(*
  Base camera system
  Implements I_Camera: set I_CameraSink.   
*)
FUNCTION_BLOCK ABSTRACT FB_CameraBase EXTENDS FB_Commons IMPLEMENTS I_Camera, I_CameraTriggerDevice

VAR
  _bInitialized             : BOOL;
  _iCameraSink              : I_CameraSink;
  _iCameraTrigger           : I_CameraTrigger;
  _bSimulate                : BOOL;
  _nPrintUnitResolution     : UDINT;           (*printhead pixel resolution [dpi]*)
  _nPrintUnitSubPx          : UDINT;           (*print unit SubPixel resolution [SubPx]*)
  _bUseCameraTrigger        : BOOL;            (*use a trigger output timestamp I/O*)
  _bUseCameraTriggerFeedback : BOOL;           (*use a camera triggered feedback timestamp I/O*)
  _eCameraMode              : E_CameraMode;    (*desired camera mode*)
  _ePossibleMode            : E_CameraMode;    (*currently possible mode*)
  _fSubstrateLength         : LREAL := 1;      (*Substrate length [m]*)
  _fSubstrateWidth          : LREAL := 1;      (*Substrate width [m]*)
  _fImageLength             : LREAL := 1;      (*Image length [m]*)
  _fImageWidth              : LREAL := 1;      (*Image width [m]*)
  _fFrameLength             : LREAL := 1;      (*Camera Frame width in [px]*)
  _bActivated               : BOOL;            (*Camera is activated*)
  _sVisuName                : STRING := 'unvailable';     (*detail visualisation instance name*)
  
  // status
  _bCamTriggerOk            : BOOL;
  _bCamTriggerStarted       : BOOL;
  _bCamTriggerDone          : BOOL;   
  _nCamStartPos             : DINT;            (*Cam start position ideal [SubPx]*)
  _nCamStartPosDeviation    : DINT;            (*Cam stated position real [SubPx]*)
  _nRxCamPoints             : UDINT;           (*number of received cam points*)

  // helper
  stCamPoint                : ST_DeformationPointAccurate;(*actual camera point*)
    
  // messaging
  _pMsgConfig               : POINTER TO CalmarCommons.ST_MSG_CONFIG;
END_VAR

VAR PERSISTENT
  _fTriggerDistance         : LREAL;           (*[m] Distance between Sensor and Trigger*)
  _fTriggerPulseLength      : LREAL := 10;     (*[ms] Length of trigger signal in ms, min. 3 bus cycles*)
  _fDetectToCameraOffset    : LREAL := 0.1;    (*[m] Distance between input trigger and camera, mech.*)
  _fCameraToPrintOffset     : LREAL := 0.0;    (*[m] Distance between Camera and PU, mech, This offset can be used to shift the reference of a camera/sheet-detect, e.g. because this reference is different from to one where the alignment Camera/sheetdetect-PrintUnit has been made*)
END_VAR

METHOD ActivateCam : BOOL
VAR_INPUT
  iCameraSink : I_CameraSink;
END_VAR
IF iCameraSink = 0 THEN
  LogError('Invalid parameter (0 pointer)');
  ActivateCam := FALSE;
  RETURN; 
ELSIF _iCameraSink <> 0 AND iCameraSink <>_iCameraSink THEN
  LogError('SetSink failed: other sink already exists');
  ActivateCam := FALSE;
  RETURN; 
END_IF 

_iCameraSink := iCameraSink;
_iCameraTrigger.Enable(iCam:=THIS^, bUseCameraTrigger:=_bUseCameraTrigger, bUseCameraTriggerFeedback:=_bUseCameraTriggerFeedback);

_bActivated := TRUE;
ActivateCam:=TRUE;
END_METHOD

(*
  Activate/Deactivate camera trigger device
*)
PROPERTY bEnableTrigger : BOOL
SET
IF bEnableTrigger THEN
  _iCameraTrigger.Enable(iCam := THIS^, bUseCameraTrigger:= _bUseCameraTrigger, bUseCameraTriggerFeedback:=_bUseCameraTriggerFeedback);
ELSE
  _iCameraTrigger.Disable();
END_IF
END_SET
END_PROPERTY

(*
  Activate/Deactivate camera manual teach mode
*)
PROPERTY bManualTeach : BOOL
SET
_iCameraTrigger.bManualTeach := bManualTeach;
END_SET
END_PROPERTY

{attribute 'monitoring':='call'}
PROPERTY bSimulate : BOOL
GET
bSimulate := _bSimulate;
END_GET
SET
_bSimulate := bSimulate;
END_SET
END_PROPERTY

METHOD CamTrigger
VAR_INPUT
  bOk             : BOOL;     // trigger is ok
	nPos            : DINT;     // camera triggered position
  nPosDeviation   : DINT;     // camera started deviation
  nX0             : DINT;     // detected position sheet/repetition
END_VAR
_nRxCamPoints := 0;
_bCamTriggerStarted    := TRUE;
_bCamTriggerDone       := FALSE;
_bCamTriggerOk  := bOk;
_nCamStartPos   := nPos;
_nCamStartPosDeviation := nPosDeviation;

LogLvl(Lvl:=E_LogSeverity.Debug, Msg:=F_Concat2('CamTrigger at X0=', TO_STRING(nPos)));
IF _iCameraSink <> 0 THEN   // inform sink
  _iCameraSink.CamStarted(nX0:=nX0);
END_IF
END_METHOD

METHOD CamTriggerDone
_bCamTriggerStarted    := FALSE;  // this call marks the end of the camera trigger period
_bCamTriggerDone       := TRUE;

LogLvl(Lvl:=E_LogSeverity.Debug, Msg:='CamTriggerDone');
IF _iCameraSink <> 0 THEN   // inform sink
  _iCameraSink.CamDone();
END_IF
END_METHOD

METHOD DeactivateCam : BOOL
VAR_INPUT
  iSink : I_CameraSink;
END_VAR
IF _iCameraSink <> 0 AND iSink <> _iCameraSink THEN
  LogError('remove sink failed: inconsistent');
  DeactivateCam := FALSE;
  RETURN;  
END_IF

_iCameraSink := 0;
_iCameraTrigger.Disable();
_bActivated := FALSE;
DeactivateCam:=TRUE;
END_METHOD

{attribute 'monitoring':='call'}
PROPERTY ABSTRACT eCameraMode : E_CameraMode
GET
END_GET
END_PROPERTY

{attribute 'monitoring':='call'}
PROPERTY ABSTRACT eDeviceType : E_CameraDevice
GET
END_GET
END_PROPERTY

{attribute 'monitoring':='call'}
PROPERTY fCameraToPrintOffset : LREAL
GET
//This offset can be used to shift the reference of a camera, e.g. because this reference is different from to one where the alignment Camera-PrintUnit has been made
fCameraToPrintOffset := _fCameraToPrintOffset;
END_GET
SET
_fCameraToPrintOffset := fCameraToPrintOffset;
END_SET
END_PROPERTY

{attribute 'monitoring':='call'}
PROPERTY fDetectToCameraOffset : LREAL
GET
//This offset can be used to shift the reference of a camera, e.g. because this reference is different from to one where the alignment Camera-PrintUnit has been made
fDetectToCameraOffset := _fDetectToCameraOffset;
END_GET
SET
_fDetectToCameraOffset := fDetectToCameraOffset;
END_SET
END_PROPERTY

{attribute 'monitoring':='call'}
(* camera frame size in [px]*)
PROPERTY fFrameLength : LREAL
GET
fFrameLength := _fFrameLength;
END_GET
SET
_fFrameLength := fFrameLength;
END_SET
END_PROPERTY

{attribute 'monitoring':='call'}
(*Image Length/Depth in [m]*)
PROPERTY fImageLength : LREAL
GET
fImageLength := _fImageLength;
END_GET
SET
_fImageLength := fImageLength;
END_SET
END_PROPERTY

{attribute 'monitoring':='call'}
(*Image Width in [m]*)
PROPERTY fImageWidth : LREAL
GET
fImageWidth := _fImageWidth;
END_GET
SET
_fImageWidth := fImageWidth;
END_SET
END_PROPERTY

{attribute 'monitoring':='call'}
(*Substrate Length/Depth in [m]*)
PROPERTY fSubstrateLength : LREAL
GET
fSubstrateLength := _fSubstrateLength;
END_GET
SET
//ROI in Print direction
IF _iCameraTrigger <> 0 THEN
  _iCameraTrigger.SetSubstrateLength(fSubstrateLength := fSubstrateLength);   // save to camera trigger
  _fSubstrateLength := fSubstrateLength;                                      // save to camera
END_IF
END_SET
END_PROPERTY

{attribute 'monitoring':='call'}
(*Substrate Width in [m]*)
PROPERTY fSubstrateWidth : LREAL
GET
fSubstrateWidth := _fSubstrateWidth;
END_GET
SET
_fSubstrateWidth := fSubstrateWidth;
END_SET
END_PROPERTY

{attribute 'monitoring':='call'}
PROPERTY fTriggerDistance : LREAL
GET
fTriggerDistance := _fTriggerDistance;
END_GET
SET
_fTriggerDistance := fTriggerDistance;
END_SET
END_PROPERTY

PROPERTY fTriggerPulseLength : LREAL
GET
fTriggerPulseLength := _fTriggerPulseLength;
END_GET
END_PROPERTY

METHOD ABSTRACT GetCamStatus : BOOL
VAR_OUTPUT
  bConnectionOK  : BOOL;    // Camera connected
  bTeachOk       : BOOL;    // Teach successful
  nTeachedPoints : UDINT;   // Teached points for this job
  nScannedPoints : UDINT;   // Scanned points on current sheet  
  bCamStarted    : BOOL;    // Camera trigger is active, cam started
  bCamDone       : BOOL;    // Camera finished on last CT
  bErrors        : ARRAY[1..GVL_Camera.nC_NbCamErrors] OF BOOL;  // generic error flag list
END_VAR
END_METHOD

METHOD Init
VAR_INPUT
  nPrintUnitResolution         : UDINT;    (*printhead pixel resolution [dpi]*)
  nPrintUnitSubPx              : UDINT;    (*print unit subPixel resolution [SubPx]*)
  iCameraTrigger               : I_CameraTrigger;
  bUseCameraTrigger            : BOOL;     (*use a trigger output timestamp I/O*)
  bUseCameraTriggerFeedback    : BOOL;     (*use a camera triggered feedback timestamp I/O*)
END_VAR
IF nPrintUnitResolution <> 0 AND iCameraTrigger <> 0 THEN
  _nPrintUnitResolution := nPrintUnitResolution;
  _nPrintUnitSubPx      := nPrintUnitSubPx;
  _iCameraTrigger       := iCameraTrigger;
  
  _bUseCameraTrigger := bUseCameraTrigger;
  _bUseCameraTriggerFeedback := bUseCameraTriggerFeedback;
  
  _bInitialized := TRUE;
ELSE
  _bInitialized := FALSE;
END_IF
END_METHOD

METHOD mJobStart : BOOL
END_METHOD

(*
  Set mode to camera.
  :return: TRUE if success
*)
METHOD ABSTRACT setCameraMode : BOOL
VAR_INPUT
  eCameraMode : E_CameraMode;
END_VAR
END_METHOD

METHOD setMsgInterface : BOOL
VAR_INPUT
	pMsgConfig	: POINTER TO CalmarCommons.ST_MSG_CONFIG;
END_VAR
_pMsgConfig := pMsgConfig;
END_METHOD

{attribute 'monitoring':='call'}
PROPERTY sName : STRING
GET
sName := 'undefined';
END_GET
END_PROPERTY

{attribute 'monitoring':='call'}
PROPERTY sVisuName : STRING
GET
sVisuName := _sVisuName;
END_GET
SET
_sVisuName := sVisuName;
END_SET
END_PROPERTY

END_FUNCTION_BLOCK

(* stored: Version 1.1.0.1, ProductVersion 3.1.4024.11
   POU FB_CameraBase: Id {c8d0ba07-7a01-4a8a-a6e6-67ad2b34ba59}, SpecialFunc None
   Folder I_CameraTriggerDevice: Id {f5011c75-0834-43aa-b7e2-aca7b6c164f7}
   Method ActivateCam: Id {33bd772a-5b9c-4915-8a51-eb63f24d6151}
   Property bEnableTrigger: Id {6c3ea2f9-cfbd-47bf-bc73-a8a64d85f37d}
   Set Set: Id {bbe0ae21-ba88-43e7-9f3b-fcb04895ed56}
   Property bManualTeach: Id {2054d80c-383b-481d-81a0-644a14a4d5ad}
   Set Set: Id {72a37891-564f-4755-9c41-477a2aec5de7}
   Property bSimulate: Id {e9ee4826-75da-4464-912c-d630e20ef560}
   Get Get: Id {5d6a4cfc-736a-4062-b9b1-3d95adb4a395}
   Set Set: Id {32912b04-adf6-4d7b-9254-2821b8d2a7c1}
   Method CamTrigger: Id {c9e54620-5e47-4477-89e1-0544e896af19}
   Method CamTriggerDone: Id {fb8288bc-dd74-44a9-91c5-11369148a052}
   Method DeactivateCam: Id {a856b950-c2e0-49b9-8c57-589d4c82956d}
   Property eCameraMode: Id {f5419f48-5fc8-416b-8961-a5ce5b9602fd}
   Get Get: Id {e50c4622-1529-42ce-9864-e7bbd5630b93}
   Property eDeviceType: Id {e06b0a89-0a7d-44c8-b80b-26b03709e855}
   Get Get: Id {4535ca3f-08e0-404b-a416-d770bd58b89d}
   Property fCameraToPrintOffset: Id {647ab733-132a-4564-bd69-e5da7fa48f0a}
   Get Get: Id {67bad6d0-ab04-4bad-b252-a2f64eada85b}
   Set Set: Id {ea33a1ea-98bd-47ee-b76a-a75a4408b9a1}
   Property fDetectToCameraOffset: Id {89fc0a6f-2777-4714-88ac-113ce4abeb84}
   Get Get: Id {e3787fc9-30f7-42cf-b306-3975c5cbd8b8}
   Set Set: Id {740e8823-2efa-4a58-ae83-960d5a7f5db9}
   Property fFrameLength: Id {55652209-4cfa-4d5c-8c70-1bd64353e2e4}
   Get Get: Id {664c74cd-4f7a-4a03-a1fb-8dff67b52e22}
   Set Set: Id {9f909ab3-375b-462c-9f8e-e0d7df2240e3}
   Property fImageLength: Id {83396a01-ff57-47f5-8330-5d4582f2e532}
   Get Get: Id {273d71c6-79db-422f-a816-cb0eef0830fd}
   Set Set: Id {5eb28392-15c5-4f4b-9354-0f59ab739f0b}
   Property fImageWidth: Id {88b7930b-57bc-4faf-a474-18efec119cfa}
   Get Get: Id {12c106de-03d0-4cc7-a0ed-77fb0f695b9c}
   Set Set: Id {e21ca4b4-1e59-4cf3-84cc-bd5e7742a89b}
   Property fSubstrateLength: Id {edd4de7d-1d9c-4eb7-ac9b-28669eaf5cd9}
   Get Get: Id {0ce2f61e-5346-4c66-9a9a-ec3019d4225b}
   Set Set: Id {043cee20-d35c-4c57-80be-2c160ef2d590}
   Property fSubstrateWidth: Id {20d2452f-aba8-4817-97e6-fc10e49a2ccd}
   Get Get: Id {0512c051-81ec-41c8-87a5-d2d408ae517d}
   Set Set: Id {38fbbb3f-66ed-4862-925f-d05ec848f4f7}
   Property fTriggerDistance: Id {4240e2de-52fb-4d48-a252-b6d6fe271b86}
   Get Get: Id {eca96f48-5f88-41ff-ab23-f3d7cf5ba488}
   Set Set: Id {90087f81-8f35-46b4-8d51-6cd9020bbc07}
   Property fTriggerPulseLength: Id {79315dcf-a401-4f0f-bd02-92222f94165e}
   Get Get: Id {f5cab0bd-a79c-444f-92aa-3659fc98aa58}
   Method GetCamStatus: Id {c732e507-4da9-4243-818b-ad4dce66447e}
   Method Init: Id {f813a140-cfef-4675-8913-e7f23b490790}
   Method mJobStart: Id {16387540-3352-4e72-abbe-1245d8a82836}
   Method setCameraMode: Id {2d256e38-1ffa-4b78-a49c-ca9ba5c3a6e0}
   Method setMsgInterface: Id {4471ab02-28c1-4479-bc78-7216b66d17b1}
   Property sName: Id {477fe687-ffdf-4b57-bd1b-23b6c93d23f9}
   Get Get: Id {17fb1c31-7fee-4e3f-a38c-fe9d48801f9d}
   Property sVisuName: Id {5c77c27a-8f50-4d5a-9d47-f1d79a5105d5}
   Get Get: Id {99122080-ac83-4afd-8b42-8dfb79d502fb}
   Set Set: Id {8f1fff78-d709-4059-8cf2-bb1e890a20a6} *)
